// TIA Portal V19 export
TYPE "LEXCHANGETRAY_typeSR1000ManualCommands"
// enableManualCmds: Bool
// start: Bool
// reset: Bool
// completionClearControlBits: LEXCHANGETRAY_typeSr1000ProfinetTelegram_completionClearControlBits
// latchandErrorClearControlBits: LEXCHANGETRAY_typeSr1000ProfinetTelegram_latchandErrorClearControlBits
// operationinstructionControlBits: LEXCHANGETRAY_typeSr1000ProfinetTelegram_operationinstructionControlBits
// parameterBankNumber: LEXCHANGETRAY_typeSr1000ProfinetTelegram_parameterBankNumber
// userData128Byte: LEXCHANGETRAY_typeSr1000ProfinetTelegram_userData128Byte
// stored: Access Published
   STRUCT
      enableManualCmds : Bool;
      start : Bool;
      reset : Bool;
      completionClearControlBits : "LEXCHANGETRAY_typeSr1000ProfinetTelegram_completionClearControlBits";
      latchandErrorClearControlBits { S7_SetPoint := 'True'} : "LEXCHANGETRAY_typeSr1000ProfinetTelegram_latchandErrorClearControlBits";
      operationinstructionControlBits { S7_SetPoint := 'True'} : "LEXCHANGETRAY_typeSr1000ProfinetTelegram_operationinstructionControlBits";
      parameterBankNumber { S7_SetPoint := 'True'} : "LEXCHANGETRAY_typeSr1000ProfinetTelegram_parameterBankNumber";
      userData128Byte { S7_SetPoint := 'True'} : "LEXCHANGETRAY_typeSr1000ProfinetTelegram_userData128Byte";
   END_STRUCT;
END_TYPE
